VAR_GLOBAL PERSISTENT
	PersMachPar					: ST_MachPar;
	PersSysPar					: ST_SysPar;
END_VAR
VAR_GLOBAL CONSTANT
	MaxNrOfVacSectTakeOutUnit	: INT:= 4;	
	MAX_ZONES					: INT:= 7;
END_VAR

(* stored: Version 1.1.0.1, ProductVersion 3.1.4020.12
   GVL GVL: Id {46c3f20f-a185-49ce-ac90-9817da5d26a6} *)
